TYPE ST_ITC_MCQ :
(**************************************************************************************
 * 	Application		:	BoxControl Framework
 *	Revision		:	$Revision: 404529 $
 *	Revision date	:	$Date: 2018-04-23 08:21:38 +0200 (Mo., 23 Apr 2018) $
 *	Last changed by	:	$Author: b7bolm $
 *	URL				:	$URL: http://almscdc.swisslog.com/repo/SWPD/Development/BoxControlFramework/20_Release/trunk/01_Software/BCF/BCF/JumpStart/20_Product/10_App/11_Com/10_Lib/10_Conv/11_ITC/01_DUTs/ST_ITC_MCQ.TcDUT $
 *
 *	Purpose			:	ITC MCQ Structure
 *
 * ------------------------------------------------------------------------------------
 *	Copyright Swisslog [IP AG], Switzerland. All rights reserved.
 * 
 * ------------------------------------------------------------------------------------
 *	
 * 	Revision History: 
 *
 * 	VERSION			DATE			INITIALS			DESCRIPTION
 *	0.1				01.01.2001		swl					Example
 *
 **************************************************************************************)
STRUCT
	Position			: STRING(Conveyor.POSITION_STRINGLENGTH); // 12 Digit SIS Location MM-GGG-EEEE-FF-Z 
	Code				: INT; // 1 Digit Code 
	Speed				: BOOL; // 1 Digit Speed
	Axis1Fwd			: BOOL; // 1 Digit Axis 1 Forward 
	Axis1Rev			: BOOL; // 1 Digit Axis 1 Backward 
	Axis2Fwd			: BOOL; // 1 Digit Axis 2 Forward 
	Axis2Rev			: BOOL; // 1 Digit Axis 2 Backward 
	Axis3Fwd			: BOOL; // 1 Digit Axis 3 Forward 
	Axis3Rev			: BOOL; // 1 Digit Axis 3 Backward 
	Axis4Fwd			: BOOL; // 1 Digit Axis 4 Forward 
	Axis4Rev			: BOOL; // 1 Digit Axis 4 Backward 
	Axis5Fwd			: BOOL; // 1 Digit Axis 5 Forward 
	Axis5Rev			: BOOL; // 1 Digit Axis 5 Backward 
	Axis6Fwd			: BOOL; // 1 Digit Axis 6 Forward 
	Axis6Rev			: BOOL; // 1 Digit Axis 6 Backward 
	Button1				: BOOL; // Button
	Button2				: BOOL; // Button 
END_STRUCT
END_TYPE

(* stored: Version 1.1.0.1, ProductVersion 3.1.4022.12
   DUT ST_ITC_MCQ: Id {880ef653-3161-42ad-8e22-19742581f25c} *)
